% RSLogix 500 project I2P JOB 14 - FORWARD-REVERSE-JOG USING 3PSS 2PSS OF 1P MOTOR_BAK028.RSS, saved by version 8.30.00.16 %
PROJECT "MWL"    % processor: Bul.1763 MicroLogix 1100 Series B %

PROGRAM FILES
  LAD 2   11 rungs

DATA FILES
  O0 OUTPUT  4 elements
  I1 INPUT  6 elements
  S2 STATUS  66 elements
  B3 BINARY  2 elements
  T4 TIMER  1 elements
  C5 COUNTER  1 elements
  R6 CONTROL  1 elements
  N7 INTEGER  1 elements
  F8 FLOAT  1 elements

LADDER 2
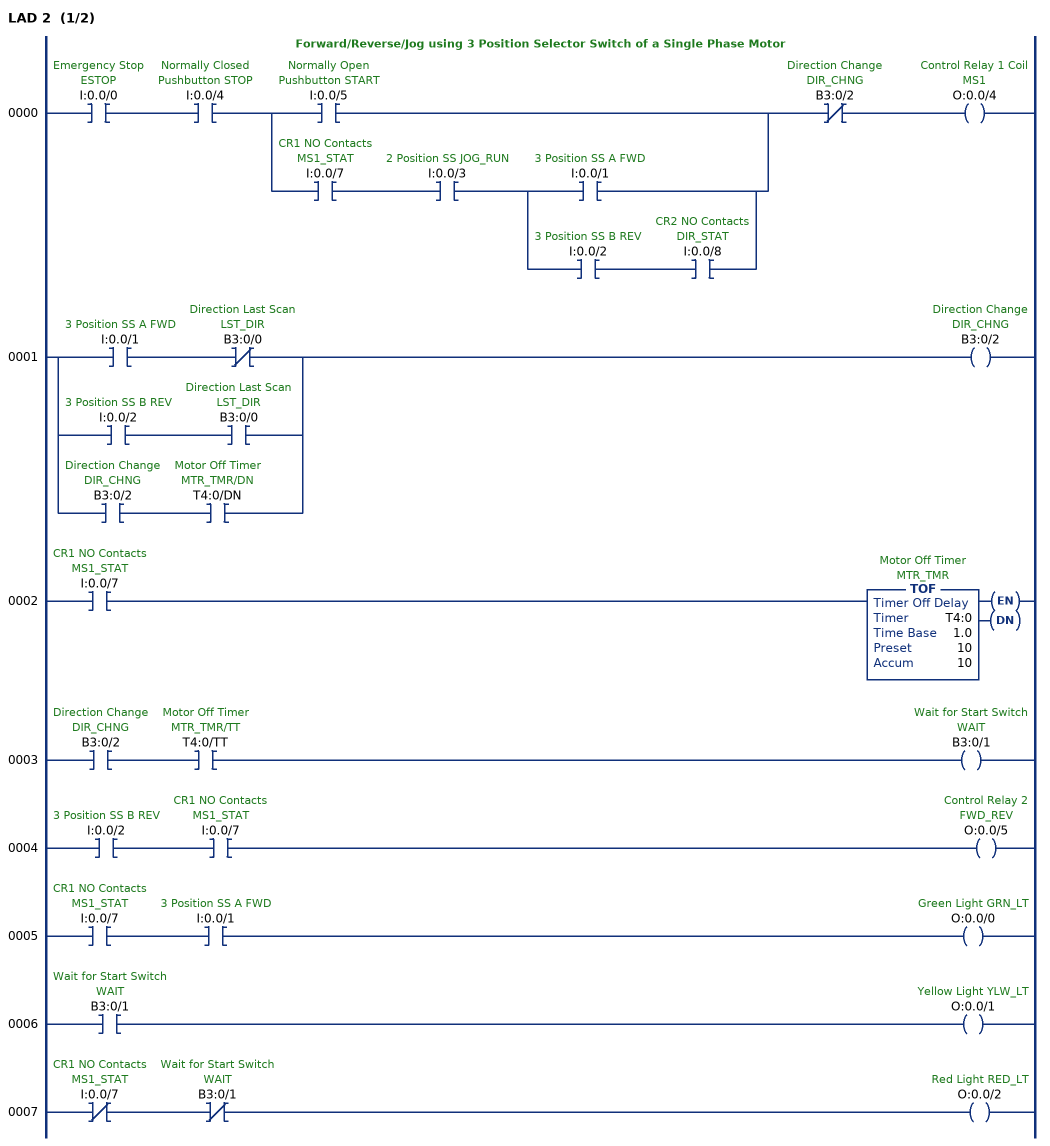
% Rung: 0 %
% TITLE: Forward/Reverse/Jog using 3 Position Selector Switch of a Single Phase Motor %
SOR XIC I:0.0/0 XIC I:0.0/4 BST XIC I:0.0/5 NXB XIC I:0.0/7 XIC I:0.0/3 BST XIC I:0.0/1 NXB XIC I:0.0/2 XIC I:0.0/8 BND BND XIO B3:0/2 OTE O:0.0/4 EOR
%   I:0.0/0  ESTOP  "Emergency Stop" %
%   I:0.0/4  STOP  "Normally Closed Pushbutton" %
%   I:0.0/5  START  "Normally Open Pushbutton" %
%   I:0.0/7  MS1_STAT  "CR1 NO Contacts" %
%   I:0.0/3  JOG_RUN  "2 Position SS" %
%   I:0.0/1  FWD  "3 Position SS A" %
%   I:0.0/2  REV  "3 Position SS B" %
%   I:0.0/8  DIR_STAT  "CR2 NO Contacts" %
%   B3:0/2  DIR_CHNG  "Direction Change" %
%   O:0.0/4  MS1  "Control Relay 1 Coil" %
% Rung: 1 %
SOR BST XIC I:0.0/1 XIO B3:0/0 NXB XIC I:0.0/2 XIC B3:0/0 NXB XIC B3:0/2 XIC T4:0/DN BND OTE B3:0/2 EOR
%   I:0.0/1  FWD  "3 Position SS A" %
%   B3:0/0  LST_DIR  "Direction Last Scan" %
%   I:0.0/2  REV  "3 Position SS B" %
%   B3:0/2  DIR_CHNG  "Direction Change" %
%   T4:0  MTR_TMR  "Motor Off Timer" %
% Rung: 2 %
SOR XIC I:0.0/7 TOF T4:0 1.0 10 10 EOR
%   I:0.0/7  MS1_STAT  "CR1 NO Contacts" %
%   T4:0  MTR_TMR  "Motor Off Timer" %
% Rung: 3 %
SOR XIC B3:0/2 XIC T4:0/TT OTE B3:0/1 EOR
%   B3:0/2  DIR_CHNG  "Direction Change" %
%   T4:0  MTR_TMR  "Motor Off Timer" %
%   B3:0/1  WAIT  "Wait for Start Switch" %
% Rung: 4 %
SOR XIC I:0.0/2 XIC I:0.0/7 OTE O:0.0/5 EOR
%   I:0.0/2  REV  "3 Position SS B" %
%   I:0.0/7  MS1_STAT  "CR1 NO Contacts" %
%   O:0.0/5  FWD_REV  "Control Relay 2" %
% Rung: 5 %
SOR XIC I:0.0/7 XIC I:0.0/1 OTE O:0.0/0 EOR
%   I:0.0/7  MS1_STAT  "CR1 NO Contacts" %
%   I:0.0/1  FWD  "3 Position SS A" %
%   O:0.0/0  GRN_LT  "Green Light" %
% Rung: 6 %
SOR XIC B3:0/1 OTE O:0.0/1 EOR
%   B3:0/1  WAIT  "Wait for Start Switch" %
%   O:0.0/1  YLW_LT  "Yellow Light" %
% Rung: 7 %
SOR XIO I:0.0/7 XIO B3:0/1 OTE O:0.0/2 EOR
%   I:0.0/7  MS1_STAT  "CR1 NO Contacts" %
%   B3:0/1  WAIT  "Wait for Start Switch" %
%   O:0.0/2  RED_LT  "Red Light" %

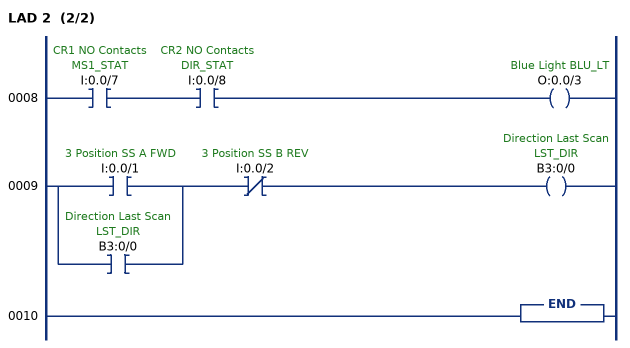
% Rung: 8 %
SOR XIC I:0.0/7 XIC I:0.0/8 OTE O:0.0/3 EOR
%   I:0.0/7  MS1_STAT  "CR1 NO Contacts" %
%   I:0.0/8  DIR_STAT  "CR2 NO Contacts" %
%   O:0.0/3  BLU_LT  "Blue Light" %
% Rung: 9 %
SOR BST XIC I:0.0/1 NXB XIC B3:0/0 BND XIO I:0.0/2 OTE B3:0/0 EOR
%   I:0.0/1  FWD  "3 Position SS A" %
%   B3:0/0  LST_DIR  "Direction Last Scan" %
%   I:0.0/2  REV  "3 Position SS B" %
% Rung: 10 %
SOR END EOR

OTHER DOCUMENTED ADDRESSES
  B3:1/0  FWD_STR
  B3:1/1  REV_STR
  I:0.0/6  PB3  "Normally Open Pushbutton"
  N7:0  LAST_DIR  "Last Direction Register"
  T4:1  STOP_TMR  "Motor Stopped Timer"

DATA TABLE (non-zero values as saved)
DATA T4
% .PRE .ACC %
% T4:0 % 10 10
